FUNCTION_BLOCK FB_CompositionBase EXTENDS FB_ComponentBase
VAR	
	aComponents					: ARRAY[0..iMaxIdxComponent] OF ITFComponent;
	eCompostitionState			: E_ComponentState;
	nComponent					: INT := -1;	
	nErrComponent				: INT;
	sErrComponentName			: STRING;
END_VAR

///
/// 
/// HF/www.asma.at/02.2018
///

PROPERTY ComponentState : E_ComponentState
GET
ComponentState := eCompostitionState;
END_GET
END_PROPERTY

PROPERTY CompostitionState : E_ComponentState
GET
CompostitionState := eCompostitionState;
END_GET
END_PROPERTY

METHOD GetComponent : POINTER TO FB_ComponentBase
VAR_INPUT
	nSubComp			:INT;	
END_VAR

VAR
	ptTmp				: POINTER TO FB_ComponentBase;
	bFound				: BOOL;
END_VAR
bFound := __QUERYPOINTER(aComponents[nSubComp], ptTmp);

IF bFound THEN
	GetComponent := ptTmp;
ELSE
	GetComponent := 0;
END_IF
END_METHOD

METHOD GetItfComponent : ITFComponent
VAR_INPUT
	nSubComp			:INT;	
END_VAR
GetItfComponent := aComponents[nSubComp];
END_METHOD

METHOD HaltAll
VAR
	iIdx			: INT;
	itfAxis			: ITFMotionComponent;
	//ptLifting		: POINTER TO FB_LiftingUnit;
END_VAR
// run all components
FOR iIdx := 0 TO GVL_CONST.iMaxIdxComponent DO
	// chk valid pointer
	IF aComponents[iIdx] <> 0 THEN
		// chk component is active
		IF NOT aComponents[iIdx].Active THEN
			CONTINUE;
		END_IF
 
		IF __QUERYINTERFACE(aComponents[iIdx], itfAxis) THEN
			itfAxis.Halt();	
		END_IF
		
	END_IF
END_FOR
END_METHOD

METHOD LoadComponents
VAR_INPUT
END_VAR
nComponent := 0;
MEMSET(ADR(aComponents), 0, SIZEOF(aComponents));
eCompostitionState := E_ComponentState.eComponentState_none;
END_METHOD

/// Registrierung von PM Sub-Komponenten.
METHOD RegisterComponent
VAR_INPUT
	ID				: INT := 0;
	fbComponent  	: ITFComponent;
END_VAR
IF fbComponent = 0 THEN
	sClearText := 'invalid sub-component pointer!';
	eCompostitionState := eComponentState_error;
	RETURN;
END_IF

// register sub-component
fbComponent.ID := ID;
fbComponent.SetEventLogReference(fbEventlog);
aComponents[nComponent] := fbComponent;

// increment counter
IF nComponent < GVL_CONST.iMaxIdxComponent THEN
	nComponent := nComponent + 1;
ELSE
	sClearText := 'max. component index overrun!';
	eCompostitionState := eComponentState_error;
	RETURN;
END_IF
END_METHOD

/// Reset component logic
{attribute 'object_name' := 'Reset'}
METHOD Reset
/// abstract base logic reset

sLastError := sEmpty;
MEMSET(ADR(stLastEvent), 0, SIZEOF(ST_EVENT));

// default: set state to ready
eState := E_ComponentState.eComponentState_ready;

/// reset all components				
ResetComponents(FALSE, FALSE, 0, 0);
END_METHOD

METHOD ResetComponents
VAR_INPUT
	bOnlyActive			: BOOL;
	bOnlyNotRunning		: BOOL;
	eComponentType		: E_ComponentType;
	eExpectType			: E_ComponentType;
END_VAR

VAR
	iIdx				: INT;
END_VAR
/// reset all components				
FOR iIdx := 0 TO GVL_CONST.iMaxIdxComponent DO
	IF aComponents[iIdx] <> 0 THEN
		
		IF aComponents[iIdx].State = eComponentState_running AND bOnlyNotRunning THEN
			CONTINUE;
		END_IF
	
		IF bOnlyActive AND NOT aComponents[iIdx].Active THEN
			CONTINUE;
		END_IF
		
		IF (eComponentType = eComponentType_none OR aComponents[iIdx].Typ = eComponentType) AND
		   (eExpectType = eComponentType_none OR aComponents[iIdx].Typ <> eExpectType) THEN
			aComponents[iIdx].Reset();		
		END_IF
		
	END_IF
END_FOR
END_METHOD

/// Run component logic
{attribute 'object_name' := 'Run'}
METHOD Run : E_ComponentState

VAR
	iIdx			: INT;
END_VAR
/// abstract base logic run

// only rdy state may lead to run
IF eState = E_ComponentState.eComponentState_ready THEN
	eState := E_ComponentState.eComponentState_running;
END_IF


// run HMI & logger
//fbEventLog.Run();

// latch resetting state
//bIsResetting := (eState = eComponentState_resetting);

/// run components

// set overall component state, prio:
// 1. E_ComponentState.eComponentState_error		( --> at least one has error)
// 2. E_ComponentState.eComponentState_none			( --> at least one state is not set)
// 3. E_ComponentState.eComponentState_resetting	( --> at least one is rsetting)
// 4. E_ComponentState.eComponentState_ready		( --> at least one is in ready state)
// 5. E_ComponentState.eComponentState_running		( --> all active are running)

// init with running state
eCompostitionState := eComponentState_running;

// run all components
FOR iIdx := 0 TO GVL_CONST.iMaxIdxComponent DO
	// chk valid pointer
	IF aComponents[iIdx] <> 0 THEN
		// chk component is active
		IF aComponents[iIdx].Active THEN
			// run component and get it's state 
			CASE aComponents[iIdx].Run() OF
				eComponentState_error:
					IF nErrComponent = 0 THEN
						nErrComponent := iIdx;
						sErrComponentName := aComponents[iIdx].Name;
					END_IF
					eCompostitionState := eComponentState_error;	
					
				eComponentState_none:
					IF eCompostitionState <> eComponentState_error THEN
						eCompostitionState := eComponentState_none;
					END_IF
					
				eComponentState_resetting:
					IF eCompostitionState <> eComponentState_error AND eCompostitionState <> eComponentState_none THEN
						eCompostitionState := eComponentState_resetting;
					END_IF
					
				eComponentState_ready:
					IF eCompostitionState = eComponentState_running THEN
						eCompostitionState := eComponentState_ready;
					END_IF					
			END_CASE
		END_IF
	END_IF
END_FOR

eState := eCompostitionState;


Run := eState;
END_METHOD

END_FUNCTION_BLOCK

(* stored: Version 1.1.0.1, ProductVersion 3.1.4022.10
   POU FB_CompositionBase: Id {26628a25-4aa5-4923-bc9b-743bc40c8134}, SpecialFunc None
   Property ComponentState: Id {884ac6f0-2a5f-4463-a592-c6513cee2658}
   Get Get: Id {1327e2aa-71a3-4e9a-8c2f-105121e18e09}
   Property CompostitionState: Id {9ebc0614-d830-4fb7-9f05-cb42458cf1e3}
   Get Get: Id {df2e4c52-4172-4ac7-9a57-490e8538e565}
   Method GetComponent: Id {42c0899e-3452-46bb-912b-b3a7f3fc85ea}
   Method GetItfComponent: Id {e2740927-c337-4beb-813f-23048662d66e}
   Method HaltAll: Id {b74779d5-a6be-47d0-954e-9123d3324930}
   Method LoadComponents: Id {fd1cb7e4-1d93-40b3-94e6-f70c9797ef8e}
   Method RegisterComponent: Id {8cf7c0b3-dc6b-4a07-94b9-9d113be3a86c}
   Method Reset: Id {1f6422c0-b152-44b0-93ad-eb6fb62f9251}
   Method ResetComponents: Id {6977f431-abb7-463b-8a67-0e1c5e31d644}
   Method Run: Id {f9d7ab07-7da4-48af-b597-c5d26c4485c9} *)
